{attribute addProperty BoxType "EJ2918-0000-0017"}
{attribute addProperty Id "FSOEAT %I*FSOE_E1AC8A65486"}
{attribute addProperty CRC "1053160623"}
{attribute addProperty SizeInBites "48"}
{attribute addProperty SizeInBytes "6"}
TYPE FSoE_Inputs_3EC5F4AF :
STRUCT
	{attribute addProperty Name "FSOE"}
	FSOE AT %I* : FSOE_E1AC8A65;
END_STRUCT
END_TYPE

(* stored: Version 1.2.0.0, ProductVersion 3.1.4024.9
   DUT FSoE_Inputs_3EC5F4AF: Id {f790ad00-1943-4f53-829b-207270cfbae4} *)
